# EPICS autosave request: basleracA130075gmApp/Db/Basler_acA1300_75gm_settings.req
## This file specifies which PVs of the corresponding database should be saved

# Enable
$(P)$(R)Enbl-Sel
# Acquisition Mode
$(P)$(R)AcqMode-Sel
# Acquisition Period
$(P)$(R)AcqPeriod-SP
# Acquisition Period Low Alarm Limit
$(P)$(R)AcqPeriodLowLim-SP
# Exposure Control Mode
$(P)$(R)ExposureMode-Sel
# Exposure Time
$(P)$(R)ExposureTime-SP
# Gain
$(P)$(R)Gain-SP
# Black Level
$(P)$(R)BlackLevel-SP
# Debouncer Period
$(P)$(R)DebouncerPeriod-SP
# Image Data Type
$(P)$(R)DataType-Sel
# Packet Size
$(P)$(R)PacketSize-SP
# Inter-Packet Delay
$(P)$(R)InterPacketDelay-SP
# Transmission Delay
$(P)$(R)TransmDelay-SP
# Bandwidth Reserve
$(P)$(R)BwReserve-SP
# Bandwidth Reserve Accumulation
$(P)$(R)BwReserveAccum-SP
# Area Of Interest Offset X
$(P)$(R)AOIOffsetX-SP
# Area Of Interest Offset Y
$(P)$(R)AOIOffsetY-SP
# Area Of Interest Width
$(P)$(R)AOIWidth-SP
# Area Of Interest Height
$(P)$(R)AOIHeight-SP
# Area Of Interest Auto Center X
$(P)$(R)AOIAutoCenterX-Sel
# Area Of Interest Auto Center X
$(P)$(R)AOIAutoCenterY-Sel
# Transformation Type
$(P)$(R)TransformType-Sel
# Multiplier for Centroid X Position Unit Convertion
$(P)$(R)ScaleFactorX-SP
# Multiplier for Centroid Y Position Unit Convertion
$(P)$(R)ScaleFactorY-SP
# Offset on image original X axis of calibration center for Centroid Position Unit Convertion
$(P)$(R)CenterOffsetX-SP
# Offset on image original Y axis of calibration center for Centroid Position Unit Convertion
$(P)$(R)CenterOffsetY-SP
# Offset of Theta for Centroid Position Unit Convertion
$(P)$(R)ThetaOffset-SP
# Real X position of calibration image center for Centroid Position Unit Convertion
$(P)$(R)CalPosCenterX-SP
# Real Y position of calibration image center for Centroid Position Unit Convertion
$(P)$(R)CalPosCenterY-SP
# Enable Background Subtraction
$(P)$(R)EnblBGSubtraction-Sel
# Enable Pixel Value Scaling and Offset
$(P)$(R)EnblOffsetScale-Sel
# Pixel Value Scale Factor
$(P)$(R)PixelScale-SP
# Pixel Value Offset
$(P)$(R)PixelOffset-SP
# Enable Low Pixel Value Clipping
$(P)$(R)EnblLowClip-Sel
# Low Clipping Value
$(P)$(R)LowClip-SP
# Enable High Pixel Value Clipping
$(P)$(R)EnblHighClip-Sel
# High Clipping Value
$(P)$(R)HighClip-SP
